(* IEC 61131-3 sources: CS_4_Aufzugsteuerung/src/Stations/CP112/Steuerung/Class/clsAntrieb, 1 file *)

(* ---- clsAntrieb.st ---- *)
(*!
<Class
	Name               = "clsAntrieb"
	Revision           = "0.0"
	RealtimeTask       = "true"
	CyclicTask         = "false"
	DefCyclictime      = "1 ms"
	BackgroundTask     = "false"
	Sigmatek           = "false"
	OSInterface        = "false"
	HighPriority       = "false"
	Automatic          = "false"
	UpdateMode         = "Prescan"
	SharedCommandTable = "true"
	Objectsize         = "(284,120)">
	<Channels>
		<Server Name="ClassSvr" Visualized="false" Initialize="false" WriteProtected="true" Retentive="false"/>
		<Server Name="sState" Visualized="true" Remotely="true" Initialize="false" WriteProtected="true" Retentive="false"/>
		<Client Name="cFahrbefehl" Required="false" Internal="false"/>
	</Channels>
</Class>
*)
clsAntrieb : CLASS
	TYPE
	  Statusautomat :
	  (
	    Stillstand:=0,
	    PowOnPos:=10,
	    FahrenPos:=20,
	    PowOnNeg:=30,
	    FahrenNeg:=40,
	    StopNormal:=99,
	    StopNot
	  )$UDINT;
	END_TYPE
  //Servers:
	ClassSvr 	: SvrChCmd_DINT;
	sState 	: SvrCh_DINT;
  //Clients:
	cFahrbefehl 	: CltChCmd_clsMotorControl;
  //Variables:
		iStep 	: Statusautomat;
		xNotStop 	: BOOL;
  //Functions:

	FUNCTION VIRTUAL GLOBAL RtWork
		VAR_INPUT
			EAX 	: UDINT;
		END_VAR
		VAR_OUTPUT
			state (EAX) 	: UDINT;
		END_VAR;

	FUNCTION GLOBAL Fahrt
		VAR_INPUT
			xDir 	: BOOL;
			xStart 	: BOOL;
		END_VAR
		VAR_OUTPUT
			xBusy 	: BOOL;
		END_VAR;

	FUNCTION GLOBAL NotAus
		VAR_INPUT
			xIn 	: BOOL;
		END_VAR;
  //Tables:
	FUNCTION @STD
		VAR_OUTPUT
			ret_code	: CONFSTATES;
		END_VAR;
	FUNCTION GLOBAL TAB @CT_;
END_CLASS;

#pragma usingLtd clsMotorControl

FUNCTION GLOBAL clsAntrieb::Fahrt
	VAR_INPUT
		xDir 	: BOOL;
		xStart 	: BOOL;
	END_VAR
	VAR_OUTPUT
		xBusy 	: BOOL;
	END_VAR

  IF xStart THEN

    IF xDir THEN
        IF (iStep <> PowOnPos) AND (iStep <> FahrenPos) THEN
            iStep := PowOnPos;
        END_IF;
    ELSE
        IF (iStep <> PowOnNeg) AND (iStep <> FahrenNeg) THEN
            iStep := PowOnNeg;
        END_IF;
    END_IF;

    xBusy := TRUE;

  ELSE

    IF iStep <> Stillstand THEN
        iStep := StopNormal;
    END_IF;

    xBusy := FALSE;

END_IF;

END_FUNCTION

FUNCTION VIRTUAL GLOBAL clsAntrieb::RtWork
	VAR_INPUT
		EAX 	: UDINT;
	END_VAR
	VAR_OUTPUT
		state (EAX) 	: UDINT;
	END_VAR

	state := READY;

  //uebergabe an HMI
  IF iStep = Stillstand THEN
    sState := 0;
  ELSIF iStep = FahrenPos THEN
    sState := 1;
  ELSIF iStep = FahrenNeg THEN
    sState := 2;
  END_IF;

  //Notstop uebergabe
  IF xNotStop THEN
    iStep := StopNot;
  END_IF;

  CASE iStep OF

      Stillstand:

          cFahrbefehl.stopNORMAL();

      PowOnPos:
          cFahrbefehl.powerOn();

          IF cFahrbefehl.sMode = clsMotorControl::MOTOR_MODE::POWER_ON THEN
              iStep := FahrenPos;
          END_IF;

      FahrenPos:
          cFahrbefehl.moveABS(position:=1215752192, velocity:=800000, acceleration:=600000);

      PowOnNeg:
          cFahrbefehl.powerOn();

          IF cFahrbefehl.sMode = clsMotorControl::MOTOR_MODE::POWER_ON THEN
              iStep := FahrenNeg;
          END_IF;

      FahrenNeg:
          cFahrbefehl.moveABS(position:=-1215752192, velocity:=800000, acceleration:=600000);

      StopNormal:
          cFahrbefehl.stopNORMAL();
          iStep := Stillstand;

      StopNot:
          cFahrbefehl.stopEMG();
          //Notstop zuruecksetzen
          IF NOT xNotStop THEN

            iStep := Stillstand;
          END_IF;

  END_CASE;

END_FUNCTION

FUNCTION GLOBAL clsAntrieb::NotAus
	VAR_INPUT
		xIn 	: BOOL;
	END_VAR

  xNotStop := xIn;

END_FUNCTION
